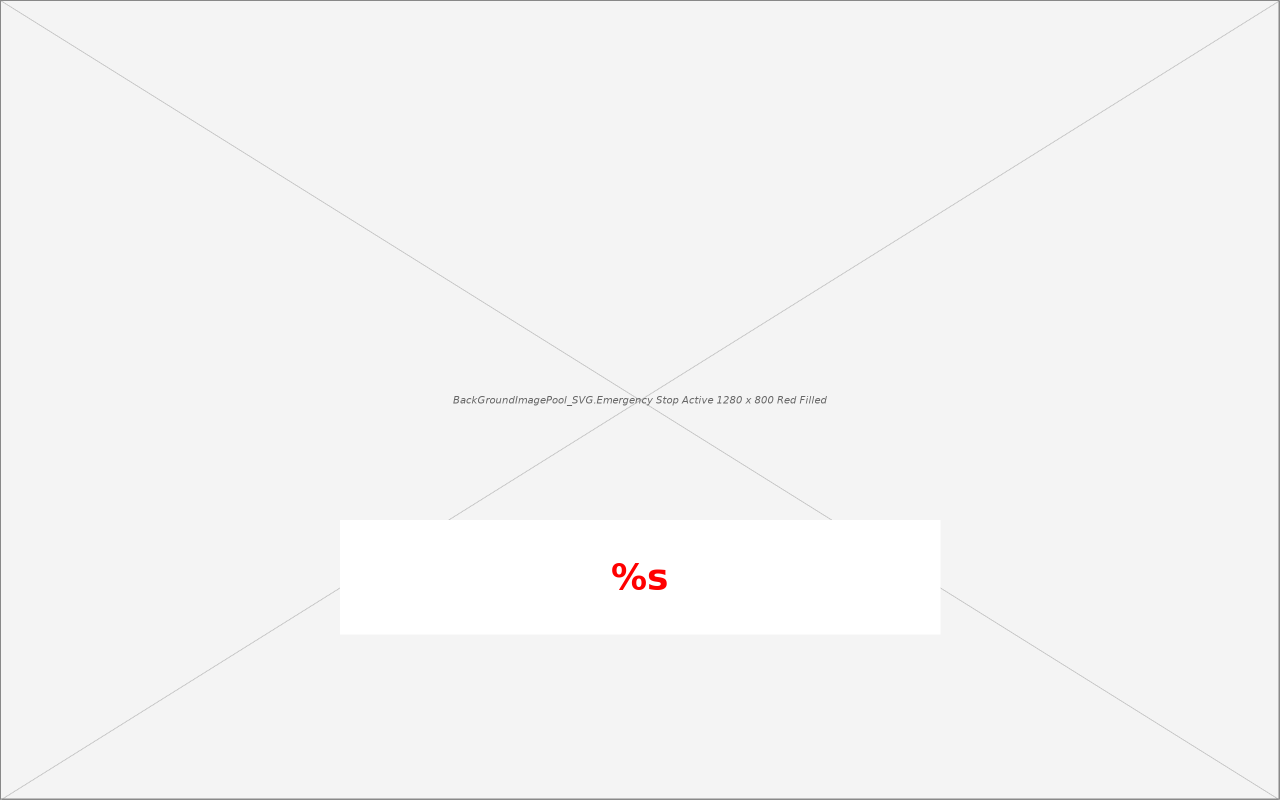
VISUALIZATION Estop  // 1280x800
VAR_IN_OUT
	bHideEstop		: BOOL ; // Hide Estop screen
END_VAR
    Image (0,0 1280x800), image: BackGroundImagePool_SVG.Emergency Stop Active 1280 x 800 Red Filled
    Textfield (340,520 600x114), "%s", text variable: GVL_HMI.sCmdEstopText
END_VISUALIZATION

(* stored: Version 1.1.0.1, ProductVersion 3.1.4024.9
   Visu Estop: Id {fb475398-f6aa-4891-8c3d-3b6fdd9b8ad0} *)
